FUNCTION_BLOCK FB_UpdateTime
VAR_INPUT
	timeToInsert:TIMESTRUCT;		(*estruta com data/hora a ser inserida*)
	actualTime:TIMESTRUCT;			(*estrutura contendo a data/hora atual*)
	bUpdateTime: BOOL;				(*atualiza a hora com um pulso nessa entrada*)
	bUpdateDate: BOOL;				(*atualiza a data com um pulso nessa entrada*)
END_VAR
VAR_OUTPUT
	bError: BOOL;						(*Erro ativo*)
	iErrorId: UDINT;					(*Id do erro*)
END_VAR
VAR
	setTime:NT_SetLocalTime;			(*Funcao para atualizar a data/hora*)
END_VAR

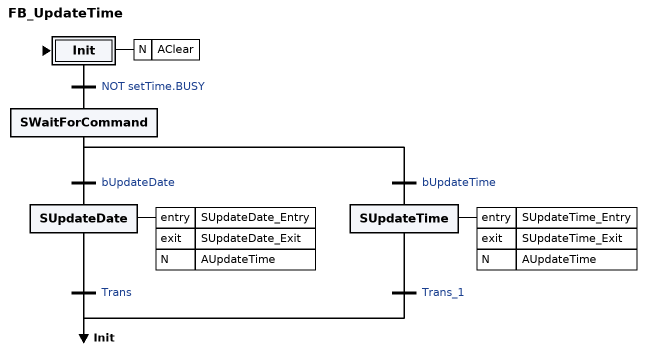
INITIAL_STEP Init:
    AClear(N);
END_STEP
TRANSITION FROM Init TO SWaitForCommand
    := NOT setTime.BUSY;
END_TRANSITION
STEP SWaitForCommand:
END_STEP
TRANSITION FROM SWaitForCommand TO SUpdateDate
    := bUpdateDate;
END_TRANSITION
STEP SUpdateDate:
    SUpdateDate_Entry(P1);  // entry action
    SUpdateDate_Exit(P0);  // exit action
    AUpdateTime(N);
END_STEP
TRANSITION FROM SUpdateDate TO Init
    := Trans;
END_TRANSITION
TRANSITION FROM SWaitForCommand TO SUpdateTime
    := bUpdateTime;
END_TRANSITION
STEP SUpdateTime:
    SUpdateTime_Entry(P1);  // entry action
    SUpdateTime_Exit(P0);  // exit action
    AUpdateTime(N);
END_STEP
TRANSITION FROM SUpdateTime TO Init
    := Trans_1;
END_TRANSITION

ACTION AClear:
setTime(	NETID:='' ,START:=FALSE );
END_ACTION

ACTION AUpdateTime:
setTime(
	NETID:='' ,
	START:= TRUE,
	ERR=>bError ,
	ERRID=> iErrorId);
END_ACTION

ACTION SUpdateDate_Entry:
(*Inicia o processo de atualizar a data*)


setTime.TIMESTR:=actualTime;
setTime.TIMESTR.wDay:=timeToInsert.wDay;
setTime.TIMESTR.wMonth:=timeToInsert.wMonth;
setTime.TIMESTR.wYear:=timeToInsert.wYear;
END_ACTION

ACTION SUpdateDate_Exit:
setTime(	NETID:='' ,START:=FALSE );
END_ACTION

ACTION SUpdateTime_Entry:
(*Inicia o processo de atualizar a data*)


setTime.TIMESTR:=actualTime;

setTime.TIMESTR.wHour:=timeToInsert.wHour;
setTime.TIMESTR.wMinute:=timeToInsert.wMinute;
setTime.TIMESTR.wSecond:=timeToInsert.wSecond;
END_ACTION

ACTION SUpdateTime_Exit:
setTime(	NETID:='' ,START:=FALSE );
END_ACTION

TRANSITION Trans:
NOT setTime.BUSY
END_TRANSITION

TRANSITION Trans_1:
NOT setTime.BUSY
END_TRANSITION

END_FUNCTION_BLOCK

(* stored: Version 1.1.0.1, ProductVersion 3.1.4020.6
   POU FB_UpdateTime: Id {ce8e0211-06d6-4438-9277-57ee5b582129}, SpecialFunc None
   Action AClear: Id {7768f2b1-763c-43a5-8435-bdea8c154ea3}
   Action AUpdateTime: Id {1f81ca51-8cab-4c3a-993e-b15271f39819}
   Action SUpdateDate_Entry: Id {f6ec4674-fb74-445a-97d3-b0f7cd40ecc3}
   Action SUpdateDate_Exit: Id {f572b11d-21b7-48fb-b850-becb8a871fa3}
   Action SUpdateTime_Entry: Id {045446b6-97a7-4f05-8076-cd018cc33d16}
   Action SUpdateTime_Exit: Id {b2eaf042-0207-4b7d-9e86-7a7068204210}
   Transition Trans: Id {75e5e0ed-d91d-46d1-9a94-4f0e6593fb8c}
   Transition Trans_1: Id {993b6255-3ca7-4a6d-9449-36d9935ea166} *)
